(* CoDeSys 2.3 project: TcpIp_SERVER_CLIENT.pro *)
(* Libraries: TcBase.lib 14.5.09 12:14:08, TcSystem.lib 21.1.15 10:22:54, STANDARD.LIB 5.6.98 12:03:02, TcpIp.lib 13.10.11 09:31:34 *)

(* Global variable list: Global_Variables *)
VAR_GLOBAL CONSTANT
	bLogDebugMessages								: BOOL := TRUE;

	MAX_CLIENT_CONNECTIONS						: UDINT(1..20) := 5;
	MAX_PLCPRJ_RXBUFFER_SIZE					: UDINT := 1000;


	PLCPRJ_RECONNECT_TIME						: TIME := T#3s;
	PLCPRJ_SEND_CYCLE_TIME						: TIME := T#1s;
	PLCPRJ_ACCEPT_POLLING_TIME					: TIME := T#1s;

	PLCPRJ_RECEIVE_POLLING_TIME		 			: TIME := T#1s;
	PLCPRJ_RECEIVE_TIMEOUT						: TIME := T#10s;

	(* Some project specific error codes *)
	PLCPRJ_ERROR_RECEIVE_BUFFER_OVERFLOW	: UDINT := 16#8101; (* receive buffer overflow*)
	PLCPRJ_ERROR_RECEIVE_TIMEOUT				: UDINT := 16#8102;(* receive timeout error *)

(*
	bLogDebugMessages								: BOOL := TRUE;

	MAX_CLIENT_CONNECTIONS						: UDINT(1..20) := 5;
	MAX_PLCPRJ_RXBUFFER_SIZE					: UDINT := 1000;


	PLCPRJ_RECONNECT_TIME						: TIME := T#3s;
(*	PLCPRJ_SEND_CYCLE_TIME						: TIME := T#1s; not used at server side *)
	PLCPRJ_ACCEPT_POLLING_TIME					: TIME := T#1s;

	PLCPRJ_RECEIVE_POLLING_TIME		 			: TIME := T#1s;
	PLCPRJ_RECEIVE_TIMEOUT						: TIME := T#50s;

	(* Some project specific error codes *)
	PLCPRJ_ERROR_RECEIVE_BUFFER_OVERFLOW	: UDINT := 16#8101; (* receive buffer overflow*)
	PLCPRJ_ERROR_RECEIVE_TIMEOUT				: UDINT := 16#8102;(* receive timeout error *)
 *)
END_VAR

(* Data type *)
TYPE E_ClientSteps :
(
	CLIENT_STATE_IDLE,
	CLIENT_STATE_CONNECT_START,
	CLIENT_STATE_CONNECT_WAIT,
	CLIENT_STATE_DATAEXCHA_START,
	CLIENT_STATE_DATAEXCHA_WAIT,
	CLIENT_STATE_CLOSE_START,
	CLIENT_STATE_CLOSE_WAIT,
	CLIENT_STATE_ERROR
);
END_TYPE

(* Data type *)
TYPE E_DataExchaSteps :
(
	DATAEXCHA_STATE_IDLE,
	DATAEXCHA_STATE_SEND_START,
	DATAEXCHA_STATE_SEND_WAIT,
	DATAEXCHA_STATE_RECEIVE_START,
	DATAEXCHA_STATE_RECEIVE_WAIT,
	DATAEXCHA_STATE_ERROR
);
END_TYPE

(* Data type *)
TYPE E_ServerSteps :
(
	SERVER_STATE_IDLE,
	SERVER_STATE_LISTENER_OPEN_START,
	SERVER_STATE_LISTENER_OPEN_WAIT,
	SERVER_STATE_REMOTE_CLIENTS_COMM,
	SERVER_STATE_REMOTE_CLIENTS_CLOSE,
	SERVER_STATE_LISTENER_CLOSE_START,
	SERVER_STATE_LISTENER_CLOSE_WAIT,
	SERVER_STATE_ERROR
);
END_TYPE

(* POU MAIN, ST *)
PROGRAM MAIN
VAR
	fbClient1						: FB_LocalClient := ( sRemoteHost:= '172.17.12.192' (* IP address of remote server!, 172.17.12.192, 172.17.36.136 *), nRemotePort:= 5000 );
	fbClient2						: FB_LocalClient := ( sRemoteHost:= '127.0.0.1', nRemotePort:= 3504 );
	fbClient3						: FB_LocalClient := ( sRemoteHost:= '127.0.0.1', nRemotePort:= 200 );
	fbClient4						: FB_LocalClient := ( sRemoteHost:= '127.0.0.1', nRemotePort:= 200 );
	fbClient5						: FB_LocalClient := ( sRemoteHost:= '127.0.0.1', nRemotePort:= 200 );

	bEnableClient1				: BOOL := FALSE;
	bEnableClient2				: BOOL := TRUE;
	bEnableClient3				: BOOL := FALSE;
	bEnableClient4				: BOOL := FALSE;
	bEnableClient5				: BOOL := FALSE;

	fbSocketCloseAll				: FB_SocketCloseAll := ( sSrvNetID := '', tTimeout := DEFAULT_ADS_TIMEOUT );
	bCloseAll					: BOOL := TRUE;

	nCount 						: UDINT;



	(* server *)
	fbServer						: FB_LocalServer := ( sLocalHost := '127.0.0.1' (*own IP address!127.17.24.129*), nLocalPort := 3504 );
	bEnableServer				: BOOL := TRUE;


END_VAR
IF bCloseAll THEN (*On PLC reset or program download close all old connections *)
	bCloseAll := FALSE;
	fbSocketCloseAll( bExecute:= TRUE );
ELSE
	fbSocketCloseAll( bExecute:= FALSE );
END_IF

IF NOT fbSocketCloseAll.bBusy THEN
	fbServer( bEnable := bEnableServer );
	nCount := nCount + 1;

	fbClient1( bEnable := bEnableClient1, sToServer := CONCAT( 'CLIENT1-', UDINT_TO_STRING( nCount ) ) );
	fbClient2( bEnable := bEnableClient2, sToServer := CONCAT( 'CLIENT2-', UDINT_TO_STRING( nCount ) ) );
	fbClient3( bEnable := bEnableClient3, sToServer := CONCAT( 'CLIENT3-', UDINT_TO_STRING( nCount ) ) );
	fbClient4( bEnable := bEnableClient4  );
	fbClient5( bEnable := bEnableClient5  );
END_IF
END_PROGRAM

(* POU Client Implementation Sample/FB_LocalClient, ST *)
FUNCTION_BLOCK FB_LocalClient
VAR_INPUT
	sRemoteHost			: STRING(15) := '127.0.0.1';(* IP adress of remote server 172.17.36.136   172.17.12.192 *)
	nRemotePort			: UDINT := 3504;
	sToServer			: T_MaxString := 'TEST';
	bEnable				: BOOL;
END_VAR
VAR_OUTPUT
	bConnected			: BOOL;
	hSocket				: T_HSOCKET;
	bBusy 				: BOOL;
	bError				: BOOL;
	nErrId				: UDINT;
	sFromServer			: T_MaxString := '';
END_VAR
VAR
	fbConnect 			: FB_SocketConnect := ( sSrvNetId := ''  );
	fbClose				: FB_SocketClose := ( sSrvNetId := '', tTimeout := DEFAULT_ADS_TIMEOUT );
	fbClientDataExcha	: FB_ClientDataExcha;

	fbConnectTON		: TON := ( PT := PLCPRJ_RECONNECT_TIME );
	fbDataExchaTON		: TON := ( PT := PLCPRJ_SEND_CYCLE_TIME );
	eStep				: E_ClientSteps;
END_VAR
CASE eStep OF

	CLIENT_STATE_IDLE:
		IF bEnable XOR bConnected THEN
			bBusy := TRUE;
			bError := FALSE;
			nErrid := 0;
			sFromServer := '';
			IF bEnable THEN
				fbConnectTON( IN := FALSE );
				eStep := CLIENT_STATE_CONNECT_START;
			ELSE
				eStep := CLIENT_STATE_CLOSE_START;
			END_IF
		ELSIF bConnected THEN
			fbDataExchaTON( IN := FALSE );
			eStep := CLIENT_STATE_DATAEXCHA_START;
		ELSE
			bBusy := FALSE;
		END_IF

	CLIENT_STATE_CONNECT_START:
		fbConnectTON( IN := TRUE, PT := PLCPRJ_RECONNECT_TIME );
		IF fbConnectTON.Q THEN
			fbConnectTON( IN := FALSE );
			fbConnect(  bExecute := FALSE  );
			fbConnect(	sRemoteHost		:= sRemoteHost,
						nRemotePort		:= nRemotePort,
						bExecute		:= TRUE );
			eStep := CLIENT_STATE_CONNECT_WAIT;
		END_IF

	CLIENT_STATE_CONNECT_WAIT:
		fbConnect( bExecute := FALSE );
		IF NOT fbConnect.bBusy THEN
			IF NOT fbConnect.bError THEN
				bConnected 	:= TRUE;
				hSocket 	:= fbConnect.hSocket;
				eStep 		:= CLIENT_STATE_IDLE;
				LogMessage( 'LOCAL client CONNECTED!', hSocket );
			ELSE
				LogError( 'FB_SocketConnect', fbConnect.nErrId );
				nErrId := fbConnect.nErrId;
				eStep := CLIENT_STATE_ERROR;
			END_IF
		END_IF

	CLIENT_STATE_DATAEXCHA_START:
		fbDataExchaTON( IN := TRUE, PT := PLCPRJ_SEND_CYCLE_TIME );
		IF fbDataExchaTON.Q THEN
			fbDataExchaTON( IN := FALSE );
			fbClientDataExcha( bExecute := FALSE );
			fbClientDataExcha( 	hSocket 	:= hSocket,
								sToServer 	:= sToServer,
								bExecute 	:= TRUE );
			eStep := CLIENT_STATE_DATAEXCHA_WAIT;
		END_IF

	CLIENT_STATE_DATAEXCHA_WAIT:
		fbClientDataExcha( bExecute := FALSE );
		IF NOT fbClientDataExcha.bBusy THEN
			IF NOT fbClientDataExcha.bError THEN
				sFromServer := fbClientDataExcha.sFromServer;
				eStep 		:= CLIENT_STATE_IDLE;
			ELSE
				(* possible errors are logged inside of fbClientDataExcha function block *)
				nErrId := fbClientDataExcha.nErrId;
				eStep :=CLIENT_STATE_ERROR;
			END_IF
		END_IF

	CLIENT_STATE_CLOSE_START:
		fbClose( bExecute := FALSE );
		fbClose(	hSocket:= hSocket,
				bExecute:= TRUE );
		eStep := CLIENT_STATE_CLOSE_WAIT;

	CLIENT_STATE_CLOSE_WAIT:
		fbClose( bExecute := FALSE );
		IF NOT fbClose.bBusy THEN
			LogMessage( 'LOCAL client CLOSED!', hSocket );
			bConnected := FALSE;
			MEMSET( ADR(hSocket), 0, SIZEOF(hSocket));
			IF fbClose.bError THEN
				LogError( 'FB_SocketClose (local client)', fbClose.nErrId );
				nErrId := fbClose.nErrId;
				eStep := CLIENT_STATE_ERROR;
			ELSE
				bBusy := FALSE;
				bError := FALSE;
				nErrId := 0;
				eStep := CLIENT_STATE_IDLE;
			END_IF
		END_IF

	CLIENT_STATE_ERROR: (* Error step *)
		bError := TRUE;
		IF bConnected THEN
			eStep := CLIENT_STATE_CLOSE_START;
		ELSE
			bBusy := FALSE;
			eStep := CLIENT_STATE_IDLE;
		END_IF
END_CASE
END_FUNCTION_BLOCK

(* POU Client Implementation Sample/FB_ClientDataExcha, ST *)
FUNCTION_BLOCK FB_ClientDataExcha
VAR_INPUT
	hSocket				: T_HSOCKET;
	sToServer			: T_MaxString;
	bExecute			: BOOL;
END_VAR
VAR_OUTPUT
	bBusy 				: BOOL;
	bError				: BOOL;
	nErrId				: UDINT;
	sFromServer			: T_MaxString;
END_VAR
VAR
	fbSocketSend		: FB_SocketSend := ( sSrvNetID := '', tTimeout := DEFAULT_ADS_TIMEOUT );
	fbSocketReceive		: FB_SocketReceive := ( sSrvNetID := '', tTimeout := DEFAULT_ADS_TIMEOUT );
	fbReceiveTON		: TON;
	fbDisconnectTON		: TON;
	RisingEdge			: R_TRIG;
	eStep				: E_DataExchaSteps;
	cbReceived, startPos, endPos, idx	: UDINT;
	cbFrame				: UDINT;
	rxBuffer				: ARRAY[0..MAX_PLCPRJ_RXBUFFER_SIZE] OF BYTE;
END_VAR
RisingEdge( CLK := bExecute );
CASE eStep OF

	DATAEXCHA_STATE_IDLE:
		IF RisingEdge.Q THEN
			bBusy := TRUE;
			bError := FALSE;
			nErrid := 0;
			fbReceiveTON( IN := FALSE, PT := T#0s ); (* don't wait, read the first answer data immediately *)
			fbDisconnectTON( IN := FALSE, PT := T#0s );(* disable timeout check first *)
			eStep := DATAEXCHA_STATE_SEND_START;
		END_IF

	DATAEXCHA_STATE_SEND_START:
		fbSocketSend( bExecute := FALSE );
		fbSocketSend( 	hSocket	:= hSocket,
						pSrc	:= ADR( sToServer ),
						cbLen	:= INT_TO_UDINT(LEN( sToServer )) + 1,(* string length inclusive zero delimiter *)
						bExecute:= TRUE );
		eStep := DATAEXCHA_STATE_SEND_WAIT;

	DATAEXCHA_STATE_SEND_WAIT:
		fbSocketSend( bExecute := FALSE );
		IF NOT fbSocketSend.bBusy THEN
			IF NOT fbSocketSend.bError THEN
				eStep := DATAEXCHA_STATE_RECEIVE_START;
			ELSE
				LogError( 'FB_SocketSend (local client)', fbSocketSend.nErrId );
				nErrId := fbSocketSend.nErrId;
				eStep := DATAEXCHA_STATE_ERROR;
			END_IF
		END_IF

	DATAEXCHA_STATE_RECEIVE_START:
		fbDisconnectTON(  );
		fbReceiveTON( IN := TRUE );
		IF fbReceiveTON.Q THEN
			fbReceiveTON( IN := FALSE );
			fbSocketReceive( bExecute := FALSE );
			fbSocketReceive(  hSocket:= hSocket,
							pDest:= ADR( rxBuffer ) + cbReceived,
							cbLen:= SIZEOF( rxBuffer ) - cbReceived,
							bExecute:= TRUE );
			eStep := DATAEXCHA_STATE_RECEIVE_WAIT;
		END_IF

	DATAEXCHA_STATE_RECEIVE_WAIT:
		fbSocketReceive( bExecute := FALSE );
		IF NOT fbSocketReceive.bBusy THEN
			IF NOT fbSocketReceive.bError THEN

				IF (fbSocketReceive.nRecBytes > 0) THEN(* bytes received *)

					startPos 		:= cbReceived;(* rxBuffer array index of first data byte *)
					endPos  		:= cbReceived + fbSocketReceive.nRecBytes  - 1;(* rxBuffer array index of last data byte *)
					cbReceived 	:= cbReceived + fbSocketReceive.nRecBytes;(* calculate the number of received data bytes *)
					cbFrame		:= 0;(* reset frame length *)

					IF cbReceived < SIZEOF( sFromServer ) THEN(* no overflow *)

						fbReceiveTON( PT := T#0s ); (* bytes received => increase the read (polling) speed *)
						fbDisconnectTON( IN := FALSE );(* bytes received => disable timeout check *)

						(* search for string end delimiter *)
						FOR idx := startPos TO endPos BY 1 DO
							IF rxBuffer[idx] = 0 THEN(* string end delimiter found *)
								cbFrame := idx + 1;(* calculate the length of the received string (inclusive the end delimiter) *)
								MEMCPY(  ADR( sFromServer ), ADR( rxBuffer ), cbFrame );(* copy the received string to the output variable (inclusive the end delimiter) *)
								MEMMOVE( ADR( rxBuffer ), ADR( rxBuffer[cbFrame] ),  cbReceived - cbFrame  );(* move the reamaining data bytes *)
								cbReceived := cbReceived - cbFrame;(* recalculate the reamaining data byte length *)
								bBusy := FALSE;
								eStep := DATAEXCHA_STATE_IDLE;
								EXIT;
							END_IF
						END_FOR

					ELSE(* there is no more free read buffer space => the answer string should be terminated *)
						LogError( 'FB_SocketReceive (local client)',  PLCPRJ_ERROR_RECEIVE_BUFFER_OVERFLOW );
						nErrId := PLCPRJ_ERROR_RECEIVE_BUFFER_OVERFLOW;(* buffer overflow !*)
						eStep := DATAEXCHA_STATE_ERROR;
					END_IF

				ELSE(* no bytes received *)
					fbReceiveTON( PT := PLCPRJ_RECEIVE_POLLING_TIME );(* no bytes received => decrease the read (polling) speed *)
					fbDisconnectTON( IN := TRUE, PT := PLCPRJ_RECEIVE_TIMEOUT );(* no bytes received => enable timeout check*)
					IF fbDisconnectTON.Q THEN (* timeout error*)
						fbDisconnectTON( IN := FALSE );
						LogError( 'FB_SocketReceive (local client)',  PLCPRJ_ERROR_RECEIVE_TIMEOUT );
						nErrID := PLCPRJ_ERROR_RECEIVE_TIMEOUT;
						eStep := DATAEXCHA_STATE_ERROR;
					ELSE(* repeat reading *)
						eStep := DATAEXCHA_STATE_RECEIVE_START; (* repeat reading *)
					END_IF
				END_IF
			ELSE(* receive error *)
				LogError( 'FB_SocketReceive (local client)',  fbSocketReceive.nErrId );
				nErrId := fbSocketReceive.nErrId;
				eStep := DATAEXCHA_STATE_ERROR;
			END_IF
		END_IF

	DATAEXCHA_STATE_ERROR:(* error step *)
		bBusy := FALSE;
		bError := TRUE;
		cbReceived := 0;
		eStep := DATAEXCHA_STATE_IDLE;

END_CASE
END_FUNCTION_BLOCK

(* POU Helper POUs/LogError, ST *)
FUNCTION LogError : DINT
VAR_INPUT
	msg			: STRING;
	nErrId		: DWORD;
END_VAR
VAR
END_VAR
IF bLogDebugMessages THEN
	IF nErrId = 0 THEN
		LogError := ADSLOGSTR( ADSLOG_MSGTYPE_HINT OR ADSLOG_MSGTYPE_LOG, CONCAT( msg, '::No error!   %s'),'' );
	ELSIF ( nErrId AND 16#80000000) =16#80000000 THEN
		LogError := ADSLOGDINT( ADSLOG_MSGTYPE_ERROR OR ADSLOG_MSGTYPE_LOG, CONCAT( msg, ':: Win32 error: %d' ), DWORD_TO_DINT(SCODE_CODE( nErrId )) );
	ELSIF (nErrId AND 16#00008100) =16#00008100 THEN
		LogError := ADSLOGDINT( ADSLOG_MSGTYPE_ERROR OR ADSLOG_MSGTYPE_LOG, CONCAT( msg, '::Internal PLC sample project error: %d' ), DWORD_TO_DINT(nErrId) );
	ELSIF (nErrId AND 16#00008000) =16#00008000 THEN
		LogError := ADSLOGDINT( ADSLOG_MSGTYPE_ERROR OR ADSLOG_MSGTYPE_LOG, CONCAT( msg, '::Internal TCP/IP Connection Server error: %d' ), DWORD_TO_DINT(nErrId) );
	ELSE
		LogError := ADSLOGDINT( ADSLOG_MSGTYPE_ERROR OR ADSLOG_MSGTYPE_LOG, CONCAT( msg, '::TwinCAT System error: %d' ), DWORD_TO_DINT(nErrId) );
	END_IF
END_IF
END_FUNCTION

(* POU Helper POUs/SCODE_CODE, ST *)
FUNCTION SCODE_CODE : DWORD
VAR_INPUT
	sc		: DWORD;
END_VAR
SCODE_CODE := 16#FFFF AND sc;
END_FUNCTION

(* POU Helper POUs/LogMessage, ST *)
FUNCTION LogMessage : DINT
VAR_INPUT
	msg		: STRING;
	hSocket	: T_HSOCKET;
END_VAR
VAR
END_VAR
IF bLogDebugMessages THEN
	LogMessage := ADSLOGDINT( ADSLOG_MSGTYPE_HINT OR ADSLOG_MSGTYPE_LOG, CONCAT( msg, '::Internal handle: %d' ), UDINT_TO_DINT(hSocket.handle)  );
END_IF
END_FUNCTION

(* POU Server Implementation Sample/FB_LocalServer, ST *)
FUNCTION_BLOCK FB_LocalServer
VAR_INPUT
	sLocalHost					: STRING(15) := '127.0.0.1';(* own IP address! *)
	nLocalPort					: UDINT := 3504;
	bEnable						: BOOL;
END_VAR
VAR_OUTPUT
	bListening					: BOOL;
	hListener 					: T_HSOCKET;
	nAcceptedClients				: UDINT;
	bBusy						: BOOL;
	bError 						: BOOL;
	nErrId						: UDINT;
END_VAR
VAR
	fbListen	 				: FB_SocketListen := ( sSrvNetID := '', tTimeout := DEFAULT_ADS_TIMEOUT );
	fbClose						: FB_SocketClose := ( sSrvNetID := '', tTimeout := DEFAULT_ADS_TIMEOUT );
	fbConnectTON				: TON := ( PT := PLCPRJ_RECONNECT_TIME );
	eStep						: E_ServerSteps;
	fbRemoteClient				: ARRAY[1..MAX_CLIENT_CONNECTIONS ] OF FB_RemoteClient;
	i							: UDINT;
END_VAR
CASE eStep OF

	SERVER_STATE_IDLE:
		IF bEnable XOR bListening THEN
			bBusy := TRUE;
			bError := FALSE;
			nErrId := 0;
			IF bEnable THEN
				fbConnectTON( IN := FALSE );
				eStep := SERVER_STATE_LISTENER_OPEN_START;
			ELSE
				eStep := SERVER_STATE_REMOTE_CLIENTS_CLOSE;
			END_IF
		ELSIF bListening THEN
			eStep := SERVER_STATE_REMOTE_CLIENTS_COMM;
		END_IF

	SERVER_STATE_LISTENER_OPEN_START:
		fbConnectTON( IN := TRUE, PT := PLCPRJ_RECONNECT_TIME );
		IF fbConnectTON.Q THEN
			fbConnectTON( IN := FALSE );
			fbListen(  bExecute := FALSE  );
			fbListen(	sLocalHost	:= sLocalHost,
					nLocalPort	:= nLocalPort,
					bExecute	:= TRUE );
			eStep := SERVER_STATE_LISTENER_OPEN_WAIT;
		END_IF

	SERVER_STATE_LISTENER_OPEN_WAIT:
		fbListen( bExecute := FALSE );
		IF NOT fbListen.bBusy THEN
			IF NOT fbListen.bError THEN
				bListening 	:= TRUE;
				hListener 	:= fbListen.hListener;
				eStep 		:= SERVER_STATE_IDLE;
				LogMessage( 'LISTENER socket OPENED!', hListener );
			ELSE
				LogError( 'FB_SocketListen',  fbListen.nErrId );
				nErrId := fbListen.nErrId;
				eStep := SERVER_STATE_ERROR;
			END_IF
		END_IF

	SERVER_STATE_REMOTE_CLIENTS_COMM:
		eStep := SERVER_STATE_IDLE;
		nAcceptedClients := 0;

		FOR i:= 1 TO MAX_CLIENT_CONNECTIONS DO
			fbRemoteClient[ i ]( hListener := hListener, bEnable := TRUE );
			IF NOT  fbRemoteClient[ i ].bBusy AND fbRemoteClient[ i ].bError THEN (*FB_SocketAccept returned error!*)
				eStep := SERVER_STATE_REMOTE_CLIENTS_CLOSE;
				EXIT;
			END_IF

			(* count the number of connected remote clients *)
			IF fbRemoteClient[ i ].bAccepted THEN
				nAcceptedClients := nAcceptedClients + 1;
			END_IF

		END_FOR

	SERVER_STATE_REMOTE_CLIENTS_CLOSE:
		nAcceptedClients := 0;
		eStep := SERVER_STATE_LISTENER_CLOSE_START; (* close listener socket too *)
		FOR i:= 1 TO MAX_CLIENT_CONNECTIONS DO
			fbRemoteClient[ i ]( bEnable := FALSE );(* close all remote client (accepted) sockets *)
			(* check if all remote client sockets are closed *)
			IF fbRemoteClient[ i ].bAccepted THEN
				eStep := SERVER_STATE_REMOTE_CLIENTS_CLOSE; (* stay here and close all remote clients first *)
				nAcceptedClients := nAcceptedClients + 1;
			END_IF
		END_FOR

	SERVER_STATE_LISTENER_CLOSE_START:
		fbClose( bExecute := FALSE );
		fbClose(	hSocket	:= hListener,
				bExecute:= TRUE );
		eStep := SERVER_STATE_LISTENER_CLOSE_WAIT;

	SERVER_STATE_LISTENER_CLOSE_WAIT:
		fbClose( bExecute := FALSE );
		IF NOT fbClose.bBusy THEN
			LogMessage( 'LISTENER socket CLOSED!', hListener );
			bListening := FALSE;
			MEMSET( ADR(hListener), 0, SIZEOF(hListener));
			IF fbClose.bError THEN
				LogError( 'FB_SocketClose (listener)',  fbClose.nErrId );
				nErrId := fbClose.nErrId;
				eStep := SERVER_STATE_ERROR;
			ELSE
				bBusy := FALSE;
				bError := FALSE;
				nErrId := 0;
				eStep := SERVER_STATE_IDLE;
			END_IF
		END_IF

	SERVER_STATE_ERROR:
		bError := TRUE;
		IF bListening THEN
			eStep := SERVER_STATE_REMOTE_CLIENTS_CLOSE;
		ELSE
			bBusy := FALSE;
			eStep := SERVER_STATE_IDLE;
		END_IF

END_CASE
END_FUNCTION_BLOCK

(* POU Server Implementation Sample/FB_RemoteClient, ST *)
FUNCTION_BLOCK FB_RemoteClient
VAR_INPUT
	hListener				: T_HSOCKET;
	bEnable 				: BOOL;
END_VAR
VAR_OUTPUT
	bAccepted			: BOOL;
	hSocket				: T_HSOCKET;
	bBusy				: BOOL;
	bError 				: BOOL;
	nErrID				: UDINT;
	sFromClient			: T_MaxString;
END_VAR
VAR
	fbAccept 			: FB_SocketAccept := ( sSrvNetID := '', tTimeout := DEFAULT_ADS_TIMEOUT );
	fbClose				: FB_SocketClose := ( sSrvNetID := '', tTimeout := DEFAULT_ADS_TIMEOUT );
	fbServerDataExcha	: FB_ServerDataExcha;
	fbAcceptTON			: TON := ( PT := PLCPRJ_ACCEPT_POLLING_TIME );
	eStep				: E_ClientSteps;
END_VAR
CASE eStep OF

	CLIENT_STATE_IDLE:
		IF bEnable XOR bAccepted THEN
			bBusy := TRUE;
			bError := FALSE;
			nErrId := 0;
			sFromClient := '';
			IF bEnable THEN
				fbAcceptTON( IN := FALSE );
				eStep := CLIENT_STATE_CONNECT_START;
			ELSE
				eStep := CLIENT_STATE_CLOSE_START;
			END_IF
		ELSIF bAccepted THEN
			eStep := CLIENT_STATE_DATAEXCHA_START;
		ELSE
			bBusy := FALSE;
		END_IF

	CLIENT_STATE_CONNECT_START:
		fbAcceptTON( IN := TRUE, PT := PLCPRJ_ACCEPT_POLLING_TIME );
		IF fbAcceptTON.Q THEN
			fbAcceptTON( IN := FALSE );
			fbAccept(  bExecute := FALSE  );
			fbAccept(	hListener := hListener,
						bExecute:= TRUE );
			eStep := CLIENT_STATE_CONNECT_WAIT;
		END_IF

	CLIENT_STATE_CONNECT_WAIT:
		fbAccept( bExecute := FALSE );
		IF NOT fbAccept.bBusy THEN
			IF NOT fbAccept.bError THEN
				IF fbAccept.bAccepted THEN
					bAccepted := TRUE;
					hSocket := fbAccept.hSocket;
					LogMessage( 'REMOTE client ACCEPTED!', hSocket );
				END_IF
				eStep := CLIENT_STATE_IDLE;
			ELSE
				LogError( 'FB_SocketAccept',  fbAccept.nErrId );
				nErrId := fbAccept.nErrId;
				eStep := CLIENT_STATE_ERROR;
			END_IF
		END_IF

	CLIENT_STATE_DATAEXCHA_START:
		fbServerDataExcha( bExecute := FALSE );
		fbServerDataExcha( 	hSocket := hSocket,
								bExecute := TRUE );
		eStep := CLIENT_STATE_DATAEXCHA_WAIT;

	CLIENT_STATE_DATAEXCHA_WAIT:
		fbServerDataExcha( bExecute := FALSE, sFromClient=>sFromClient );
		IF NOT fbServerDataExcha.bBusy THEN
			IF NOT fbServerDataExcha.bError THEN
				eStep := CLIENT_STATE_IDLE;
			ELSE
				(* possible errors are logged inside of fbServerDataExcha function block *)
				nErrId := fbServerDataExcha.nErrID;
				eStep := CLIENT_STATE_ERROR;
			END_IF
		END_IF

	CLIENT_STATE_CLOSE_START:
		fbClose( bExecute := FALSE );
		fbClose(	hSocket:= hSocket,
				bExecute:= TRUE );
		eStep := CLIENT_STATE_CLOSE_WAIT;

	CLIENT_STATE_CLOSE_WAIT:
		fbClose( bExecute := FALSE );
		IF NOT fbClose.bBusy THEN
			LogMessage( 'REMOTE client CLOSED!', hSocket );
			bAccepted := FALSE;
			MEMSET( ADR( hSocket ), 0, SIZEOF( hSocket ) );
			IF fbClose.bError THEN
				LogError( 'FB_SocketClose (remote client)', fbClose.nErrId );
				nErrId := fbClose.nErrId;
				eStep := CLIENT_STATE_ERROR;
			ELSE
				bBusy := FALSE;
				bError := FALSE;
				nErrId := 0;
				eStep := CLIENT_STATE_IDLE;
			END_IF
		END_IF

	CLIENT_STATE_ERROR:
		bError := TRUE;
		IF bAccepted THEN
			eStep := CLIENT_STATE_CLOSE_START;
		ELSE
			eStep := CLIENT_STATE_IDLE;
			bBusy := FALSE;
		END_IF

END_CASE
END_FUNCTION_BLOCK

(* POU Server Implementation Sample/FB_ServerDataExcha, ST *)
FUNCTION_BLOCK FB_ServerDataExcha
VAR_INPUT
	hSocket			: T_HSOCKET;
	bExecute		: BOOL;
END_VAR
VAR_OUTPUT
	bBusy			: BOOL;
	bError 			: BOOL;
	nErrID			: UDINT;
	sFromClient		: T_MaxString;
END_VAR
VAR
	fbSocketReceive	: FB_SocketReceive := ( sSrvNetId := '', tTimeout := DEFAULT_ADS_TIMEOUT );
	fbSocketSend	: FB_SocketSend :=  ( sSrvNetId := '', tTimeout := DEFAULT_ADS_TIMEOUT );
	eStep			: E_DataExchaSteps;
	RisingEdge		: R_TRIG;
	fbReceiveTON	: TON;
	fbDisconnectTON 	: TON;
	cbReceived, startPos, endPos, idx	: UDINT;
	cbFrame			: UDINT;
	rxBuffer			: ARRAY[0..MAX_PLCPRJ_RXBUFFER_SIZE] OF BYTE;
END_VAR
RisingEdge( CLK := bExecute );
CASE eStep OF

	DATAEXCHA_STATE_IDLE:
		IF RisingEdge.Q THEN
			bBusy 	:= TRUE;
			bError 	:= FALSE;
			nErrId 	:= 0;
			fbDisconnectTON( IN := FALSE, PT := T#0s );(* disable timeout check first *)
			fbReceiveTON( IN := FALSE, PT := T#0s ); (* receive first request immediately *)
			eStep 	:= DATAEXCHA_STATE_RECEIVE_START;
		END_IF

	DATAEXCHA_STATE_RECEIVE_START: (* Receive remote client data *)
		fbReceiveTON(  IN := TRUE );
		IF fbReceiveTON.Q THEN
			fbReceiveTON( IN := FALSE );
			fbSocketReceive( bExecute := FALSE );
			fbSocketReceive( 	hSocket		:= hSocket,
							pDest		:= ADR( rxBuffer ) + cbReceived,
							cbLen		:= SIZEOF( rxBuffer ) - cbReceived,
							bExecute	:= TRUE );
			eStep := DATAEXCHA_STATE_RECEIVE_WAIT;
		END_IF

	DATAEXCHA_STATE_RECEIVE_WAIT:
		fbSocketReceive( bExecute := FALSE );
		IF NOT fbSocketReceive.bBusy THEN
			IF NOT fbSocketReceive.bError THEN

				IF (fbSocketReceive.nRecBytes > 0) THEN(* bytes received *)

					startPos 		:= cbReceived;(* rxBuffer array index of first data byte *)
					endPos  		:= cbReceived + fbSocketReceive.nRecBytes  - 1;(* rxBuffer array index of last data byte *)
					cbReceived 	:= cbReceived + fbSocketReceive.nRecBytes;(* calculate the number of received data bytes *)
					cbFrame		:= 0;(* reset frame length *)

					IF cbReceived < SIZEOF( sFromClient ) THEN(* no overflow *)

						fbReceiveTON( IN := FALSE, PT := T#0s ); (* bytes received => increase the read (polling) speed *)
						fbDisconnectTON( IN := FALSE, PT := PLCPRJ_RECEIVE_TIMEOUT );(* bytes received => disable timeout check *)

						(* search for string end delimiter *)
						FOR idx := startPos TO endPos BY 1 DO
							IF rxBuffer[idx] = 0 THEN(* string end delimiter found *)
								cbFrame := idx + 1;(* calculate the length of the received string (inclusive the end delimiter) *)
								MEMCPY(  ADR( sFromClient ), ADR( rxBuffer ), cbFrame );(* copy the received string to the output variable (inclusive the end delimiter) *)
								MEMMOVE( ADR( rxBuffer ), ADR( rxBuffer[cbFrame] ),  cbReceived - cbFrame  );(* move the reamaining data bytes *)
								cbReceived := cbReceived - cbFrame;(* recalculate the reamaining data byte length *)
								eStep := DATAEXCHA_STATE_SEND_START;
								EXIT;
							END_IF
						END_FOR

					ELSE(* there is no more free read buffer space => the answer string should be terminated *)
						LogError( 'FB_SocketReceive (remote client)',  PLCPRJ_ERROR_RECEIVE_BUFFER_OVERFLOW );
						nErrId := PLCPRJ_ERROR_RECEIVE_BUFFER_OVERFLOW;(* buffer overflow !*)
						eStep := DATAEXCHA_STATE_ERROR;
					END_IF

				ELSE(* no bytes received *)
					fbReceiveTON( IN := FALSE, PT := PLCPRJ_RECEIVE_POLLING_TIME );(* no bytes received => decrease the read (polling) speed *)
					fbDisconnectTON( IN := TRUE, PT := PLCPRJ_RECEIVE_TIMEOUT );(* no bytes received => enable timeout check*)
					IF fbDisconnectTON.Q THEN (* timeout error*)
						fbDisconnectTON( IN := FALSE );
						LogError( 'FB_SocketReceive (remote client)',  PLCPRJ_ERROR_RECEIVE_TIMEOUT );
						nErrID := PLCPRJ_ERROR_RECEIVE_TIMEOUT;
						eStep := DATAEXCHA_STATE_ERROR;
					ELSE(* repeat reading *)
						eStep := DATAEXCHA_STATE_RECEIVE_START; (* repeat reading *)
					END_IF
				END_IF
			ELSE(* receive error *)
				LogError( 'FB_SocketReceive (remote client)',  fbSocketReceive.nErrId );
				nErrId := fbSocketReceive.nErrId;
				eStep := DATAEXCHA_STATE_ERROR;
			END_IF
		END_IF

	DATAEXCHA_STATE_SEND_START:
		fbSocketSend( bExecute := FALSE );
		fbSocketSend(	hSocket	:= hSocket,
						pSrc	:= ADR( sFromClient ),
						cbLen	:= INT_TO_UDINT(LEN( sFromClient )) + 1,(* string length inclusive the zero delimiter *)
						bExecute:= TRUE );
		eStep := DATAEXCHA_STATE_SEND_WAIT;

	DATAEXCHA_STATE_SEND_WAIT:
		fbSocketSend( bExecute := FALSE );
		IF NOT fbSocketSend.bBusy THEN
			IF NOT fbSocketSend.bError THEN
				bBusy := FALSE;
				eStep := DATAEXCHA_STATE_IDLE;
			ELSE
				LogError( 'fbSocketSend (remote client)',  fbSocketSend.nErrId );
				nErrId := fbSocketSend.nErrId;
				eStep := DATAEXCHA_STATE_ERROR;
			END_IF
		END_IF

	DATAEXCHA_STATE_ERROR:
		bBusy := FALSE;
		bError := TRUE;
		cbReceived := 0;(* reset old received data bytes *)
		eStep := DATAEXCHA_STATE_IDLE;
END_CASE
END_FUNCTION_BLOCK

(* POU MAIN_SERVER, ST *)
PROGRAM MAIN_SERVER
VAR
	fbServer						: FB_LocalServer := ( sLocalHost := '127.0.0.1' (*own IP address!127.17.24.129*), nLocalPort := 3504 );
	bEnableServer				: BOOL := TRUE;
	fbSocketCloseAll				: FB_SocketCloseAll :=  ( sSrvNetID := '', tTimeout := DEFAULT_ADS_TIMEOUT );
	bCloseAll					: BOOL := TRUE;
END_VAR
IF bCloseAll THEN (*On PLC reset or program download close all old connections *)
	bCloseAll := FALSE;
	fbSocketCloseAll( bExecute:= TRUE );
ELSE
	fbSocketCloseAll( bExecute:= FALSE );
END_IF

IF NOT fbSocketCloseAll.bBusy THEN
	fbServer( bEnable := bEnableServer );
END_IF
END_PROGRAM
